(* IEC 61131-3 sources: Industrial-Meter-Tracking-System-Modernization/plc/global, 2 files *)

(* ---- history-struct.st ---- *)
(*
    Type: History
    Purpose:
    Stores production state snapshot for later transfer to SCADA / SQL.

    Note:
    This is an anonymized version of the original structure.
*)

TYPE History :
STRUCT
    NotTransferred_Server1 : BOOL;
    NotTransferred_Server2 : BOOL;
    NotTransferred_Server3 : BOOL;
    NotTransferred_Server4 : BOOL;

    ShiftNumber   : WORD;
    OrderNumber   : DWORD;

    InputCounter  : DWORD;
    OutputCounter : DWORD;
    RejectCounter : DWORD;

    Year          : WORD;
    Month         : WORD;
    Day           : WORD;
    Hour          : WORD;
    Minute        : WORD;
    Second        : WORD;

    StatusWord    : WORD;
    StatusWord2   : WORD;

    UserNumber    : WORD;
    SetupType     : WORD;
END_STRUCT
END_TYPE

(* ---- gvl-example.st ---- *)
(*
    Global Variables Example
    Purpose:
    Shows the main categories of global variables used in the PLC project.

    Real memory addresses, line names and internal identifiers were removed.
*)

VAR_GLOBAL RETAIN

    // Shift and time
    PreviousScanShift : WORD;
    CurrentShift      : WORD;

    CurrentYear       : WORD;
    CurrentMonth      : WORD;
    CurrentDay        : WORD;
    CurrentHour       : WORD;
    CurrentMinute     : WORD;
    CurrentSecond     : WORD;

    // Line status
    LineStatusWord    : WORD;
    LineStatusWord2   : WORD;
    PanelButtonsWord  : WORD;

    // Production counters
    CurrentOrderCounter : DWORD;
    GlobalShiftCounter  : DWORD;
    OrderNumber         : DWORD;

    // Transfer handshake
    DataNeedSendToServer1 : WORD; // 0 = ready, 1 = data prepared, 2 = server confirmed
    DataNeedSendToServer2 : WORD;

    // History transfer buffer
    HistYear          : WORD;
    HistMonth         : WORD;
    HistDay           : WORD;
    HistHour          : WORD;
    HistMinute        : WORD;
    HistSecond        : WORD;

    HistInputCounter  : DWORD;
    HistOutputCounter : DWORD;
    HistRejectCounter : DWORD;
    HistOrderNumber   : DWORD;
    HistStatusWord    : WORD;
    HistShiftNumber   : WORD;

    // Roll / meter counters
    Roll1Meters       : DWORD;
    Roll2Meters       : DWORD;
    Roll3Meters       : DWORD;
    Roll4Meters       : DWORD;
    Roll5Meters       : DWORD;
    FinalProductMeters: DWORD;

    // Values prepared for sending
    SendRoll1Meters   : DWORD;
    SendRoll2Meters   : DWORD;
    SendRoll3Meters   : DWORD;
    SendRoll4Meters   : DWORD;
    SendRoll5Meters   : DWORD;

    // Modbus diagnostics
    ModbusErrorsWord  : WORD;
    ModbusResetWord   : WORD;

END_VAR

VAR_GLOBAL
    LineHistory : ARRAY[1..20000] OF History;
END_VAR
